// Mitsubishi GX Works2 project: project 1 auto   PLC: FX3G

// global labels: Global1
VAR_GLOBAL
  Starter AT X010 : BOOL;
  WorkDay_Lamp AT Y010 : BOOL;
  Emergancy AT X007 : BOOL;
  Invalid_Stock AT M0 : BOOL;
  Flour_Stock AT D1600 : REAL;
END_VAR
VAR_GLOBAL CONSTANT
  Const_100 : REAL := 100;
END_VAR
VAR_GLOBAL
  Yeast_Stock AT D1610 : REAL;
END_VAR
VAR_GLOBAL CONSTANT
  const_yeast_5 : REAL := 5.0;
END_VAR
VAR_GLOBAL
  Yeast_Div AT D1615 : REAL;
  Water_Stock AT D1620 : REAL;
  Water_Div AT D1625 : REAL;
END_VAR
VAR_GLOBAL CONSTANT
  Const_Water_2 : REAL := 2;
END_VAR
VAR_GLOBAL
  Oil_Stock AT D1630 : REAL;
  Oil_Div AT D1635 : REAL;
END_VAR
VAR_GLOBAL CONSTANT
  Oil_const : REAL := 3.33333333;
END_VAR
VAR_GLOBAL
  Spicies_Stock AT D1640 : REAL;
  Spicies_Div AT D1645 : REAL;
END_VAR
VAR_GLOBAL CONSTANT
  Const_Spicies_10 : REAL := 10;
  Const_3_Sec : INT := 30;
END_VAR
VAR_GLOBAL
  Start_Move AT X002 : BOOL;
  checkKK AT TS0 : BOOL;
  Lamp_Y5 AT Y005 : BOOL;
  Timer_In AT TC0 : BOOL;
END_VAR
VAR_GLOBAL CONSTANT
  TIMERINN : INT := 30;
END_VAR
VAR_GLOBAL
  check_y05 AT TS0 : BOOL;
  check_lamp5 AT M2 : BOOL;
  checkM2 AT M2 : BOOL;
  Input_X1 AT X001 : BOOL;
  Lamp_Y1 AT Y001 : BOOL;
  Start_Stage_2 AT X011 : BOOL;
  Couner_X11 AT CC2 : BOOL;
END_VAR
VAR_GLOBAL CONSTANT
  Max_11 : INT := 2;
END_VAR
VAR_GLOBAL
  Check_Counter_x11 AT CS2 : BOOL;
  Timer_Y002 AT TC1 : BOOL;
END_VAR
VAR_GLOBAL CONSTANT
  Max_Time_Y002 : INT := 10;
END_VAR
VAR_GLOBAL
  Check_Lights AT M3 : BOOL;
  Check_Y002 AT TS1 : BOOL;
  Lamp_Y2 AT Y002 : BOOL;
  Timer_Y003 AT TC2 : BOOL;
END_VAR
VAR_GLOBAL CONSTANT
  Max_Time_Y003 : INT := 10;
END_VAR
VAR_GLOBAL
  Check_Y003 AT TS2 : BOOL;
  Lamp_Y003 AT Y003 : BOOL;
END_VAR
VAR_GLOBAL CONSTANT
  Total_Time_stage2 : INT := 30;
END_VAR
VAR_GLOBAL
  Timer_Total AT TC3 : BOOL;
  Timer_Total_Ending AT TS3 : BOOL;
  Timer_Y004 AT TC4 : BOOL;
END_VAR
VAR_GLOBAL CONSTANT
  Max_Time_Y004 : INT := 40;
END_VAR
VAR_GLOBAL
  Y004_Open AT TS4 : BOOL;
  Baking_Lamp AT Y004 : BOOL;
  Check_Stage2_End AT M4 : BOOL;
  Close_Y004 AT TS4 : BOOL;
  Start_Check_Quality AT X003 : BOOL;
  Input_Analog_Value AT D8281 : REAL;
END_VAR
VAR_GLOBAL CONSTANT
  Const_2000 : DINT := 2000;
  Const_400 : DINT := 400;
END_VAR
VAR_GLOBAL
  Check_Quality_Status AT M5 : BOOL;
  Check_Quality_Value AT M5 : BOOL;
  Check_Quality_Fail AT M5 : BOOL;
  Quality_Lamp AT Y006 : BOOL;
  Check_Successful AT TS5 : BOOL;
  Check6 AT M6 : BOOL;
  Timer_Y006 AT TC5 : BOOL;
END_VAR
VAR_GLOBAL CONSTANT
  Max_Time_YOO5 : INT := 50;
END_VAR
VAR_GLOBAL
  stop_Y006 AT TS5 : BOOL;
  analog AT D8281 : WORD;
  analogResolt AT D1700 : DINT;
  y6_lamp AT Y006 : BOOL;
END_VAR
VAR_GLOBAL CONSTANT
  Max_Time_YOO6 : INT := 50;
END_VAR
VAR_GLOBAL
  Flower_Tank AT D1650 : REAL;
  Yeast_Tank AT D1655 : REAL;
  Water_Tank AT D1660 : REAL;
  Oil_Tank AT D1665 : REAL;
  Spicies_Tank AT D1670 : REAL;
  Lisha AT M1 : BOOL;
  Flower_In_Mixer AT D1675 : REAL;
  Yeast_In_Mixer AT D1680 : REAL;
  Water_In_Mixer AT D1685 : REAL;
  Oil_In_Mixer AT D1690 : REAL;
  Spicies_In_Mixer AT D1695 : REAL;
  Flower_In_Blow AT D1705 : REAL;
  Yeast_In_Blow AT D1710 : REAL;
  Water_In_Blow AT D1715 : REAL;
  Oil_In_Blow AT D1720 : REAL;
  Spicies_In_Blow AT D1725 : REAL;
END_VAR
VAR_GLOBAL CONSTANT
  Const_20 : REAL := 20;
  Const_50 : REAL := 50;
  Const_30 : REAL := 30;
  Const_10 : REAL := 10;
END_VAR
VAR_GLOBAL
  Flour_Resolt AT D1730 : REAL;
  Yeast_Result AT D1735 : REAL;
  Water_Result AT D1740 : REAL;
  Oil_Result AT D1745 : REAL;
  Spieces_Result AT D1750 : REAL;
  Flower_In_Pattern AT D1755 : REAL;
  Yeast_In_Pattern AT D1760 : REAL;
  Water_In_Pattern AT D1765 : REAL;
  Oil_In_Pattern AT D1770 : REAL;
  Spicies_In_Pattern AT D1780 : REAL;
  Counter_M5 AT CC5 : BOOL;
END_VAR
VAR_GLOBAL CONSTANT
  Max_M5 : INT := 2;
END_VAR
VAR_GLOBAL
  Drop_Pattern AT CS5 : BOOL;
  Dropping_Time AT TC6 : BOOL;
END_VAR
VAR_GLOBAL CONSTANT
  Max_Drop_Time : INT := 30;
END_VAR
VAR_GLOBAL
  Stop_Y10 AT TS6 : BOOL;
  Check_3_Lights AT M7 : BOOL;
  Timer_Y010 AT TC10 : BOOL;
END_VAR
VAR_GLOBAL CONSTANT
  Max_Time_Y010 : INT := 5;
END_VAR
VAR_GLOBAL
  stop_timerY10 AT TS10 : BOOL;
  Check_X10 AT M10 : BOOL;
  Start_Check_Quuality AT X003 : BOOL;
  Check_Light10 AT M10 : BOOL;
  Timer_Y010_Close AT TC11 : BOOL;
  Stop_3_sconds_y10 AT TS6 : BOOL;
  open_y10 AT M11 : BOOL;
  stop_timerY100 AT TS11 : BOOL;
  TRY AT M12 : BOOL;
  yosi AT M13 : BOOL;
  jwegfw AT M13 : BOOL;
  G AT M20 : BOOL;
END_VAR
VAR_GLOBAL CONSTANT
  Max_Time_Y01000 : INT := 5;
END_VAR
VAR_GLOBAL
  fictivy AT Y020 : BOOL;
  Shut_Down_Y10 AT M13 : BOOL;
  Start_New_Itaration AT M14 : BOOL;
  Invalid_Stock_Next_Itaration AT M15 : BOOL;
  notgood AT M16 : BOOL;
END_VAR

// task Task_01 (event TRUE, interval 0, priority 31): POU_01

PROGRAM POU_01
(* structured ladder/FBD written out as ST: instructions are called as NAME(EN, inputs, outputs); _pN, _eN, _tN stand for wires *)
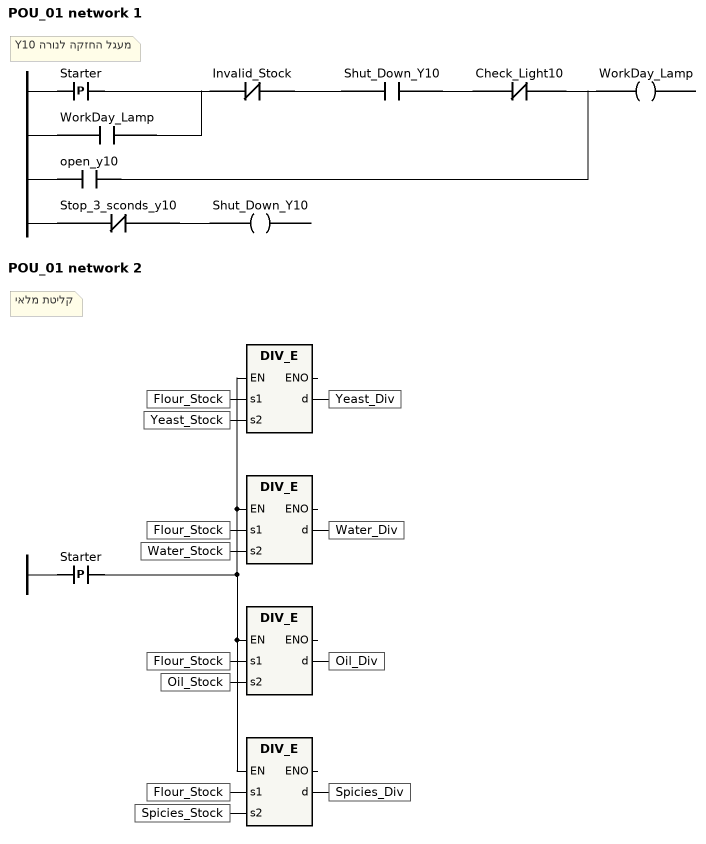
(* network 1 מעגל החזקה לנורה Y10 *)
(* מעגל החזקה לנורה Y10 *)
WorkDay_Lamp := ((((LDP(TRUE, Starter) OR WorkDay_Lamp) AND NOT Invalid_Stock) AND Shut_Down_Y10) AND NOT Check_Light10) OR open_y10;
Shut_Down_Y10 := NOT Stop_3_sconds_y10;
(* network 2 קליטת וחישוב מלאי *)
(* קליטת מלאי *)
_p1 := LDP(TRUE, Starter);
DIV_E(_p1, Flour_Stock, Yeast_Stock, Yeast_Div);
DIV_E(_p1, Flour_Stock, Water_Stock, Water_Div);
DIV_E(_p1, Flour_Stock, Oil_Stock, Oil_Div);
DIV_E(_p1, Flour_Stock, Spicies_Stock, Spicies_Div);
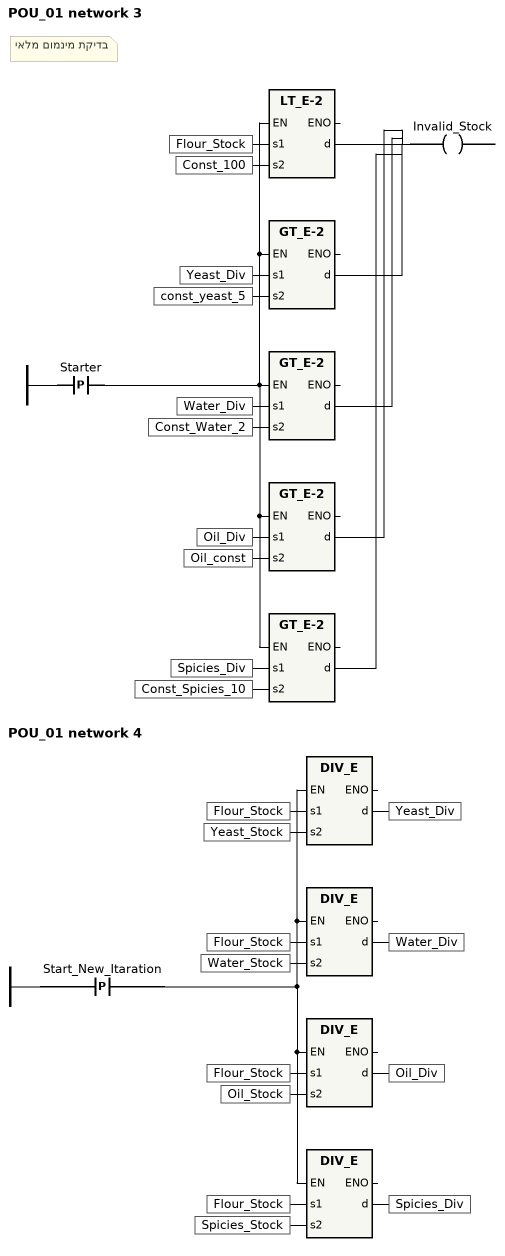
(* network 3 בדיקת מינימום מלאי *)
(* בדיקת מינמום מלאי *)
_p1 := LDP(TRUE, Starter);
LT_E(_p1, Flour_Stock, Const_100, _t2);
GT_E(_p1, Yeast_Div, const_yeast_5, _t3);
GT_E(_p1, Water_Div, Const_Water_2, _t4);
GT_E(_p1, Oil_Div, Oil_const, _t5);
GT_E(_p1, Spicies_Div, Const_Spicies_10, _t6);
Invalid_Stock := _t2 OR _t3 OR _t4 OR _t5 OR _t6;
(* network 4 בדיקת מלאי נוספת *)
_p1 := LDP(TRUE, Start_New_Itaration);
DIV_E(_p1, Flour_Stock, Yeast_Stock, Yeast_Div);
DIV_E(_p1, Flour_Stock, Water_Stock, Water_Div);
DIV_E(_p1, Flour_Stock, Oil_Stock, Oil_Div);
DIV_E(_p1, Flour_Stock, Spicies_Stock, Spicies_Div);
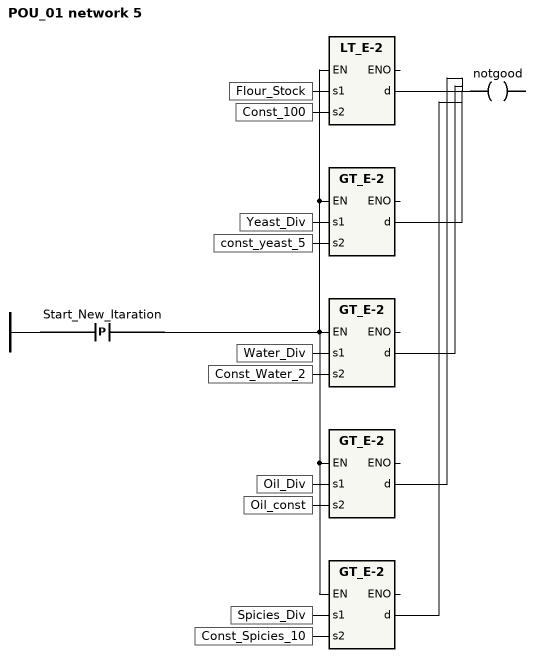
(* network 5 בדיקת מלאי נוספת *)
_p1 := LDP(TRUE, Start_New_Itaration);
LT_E(_p1, Flour_Stock, Const_100, _t2);
GT_E(_p1, Yeast_Div, const_yeast_5, _t3);
GT_E(_p1, Water_Div, Const_Water_2, _t4);
GT_E(_p1, Oil_Div, Oil_const, _t5);
GT_E(_p1, Spicies_Div, Const_Spicies_10, _t6);
notgood := _t2 OR _t3 OR _t4 OR _t5 OR _t6;
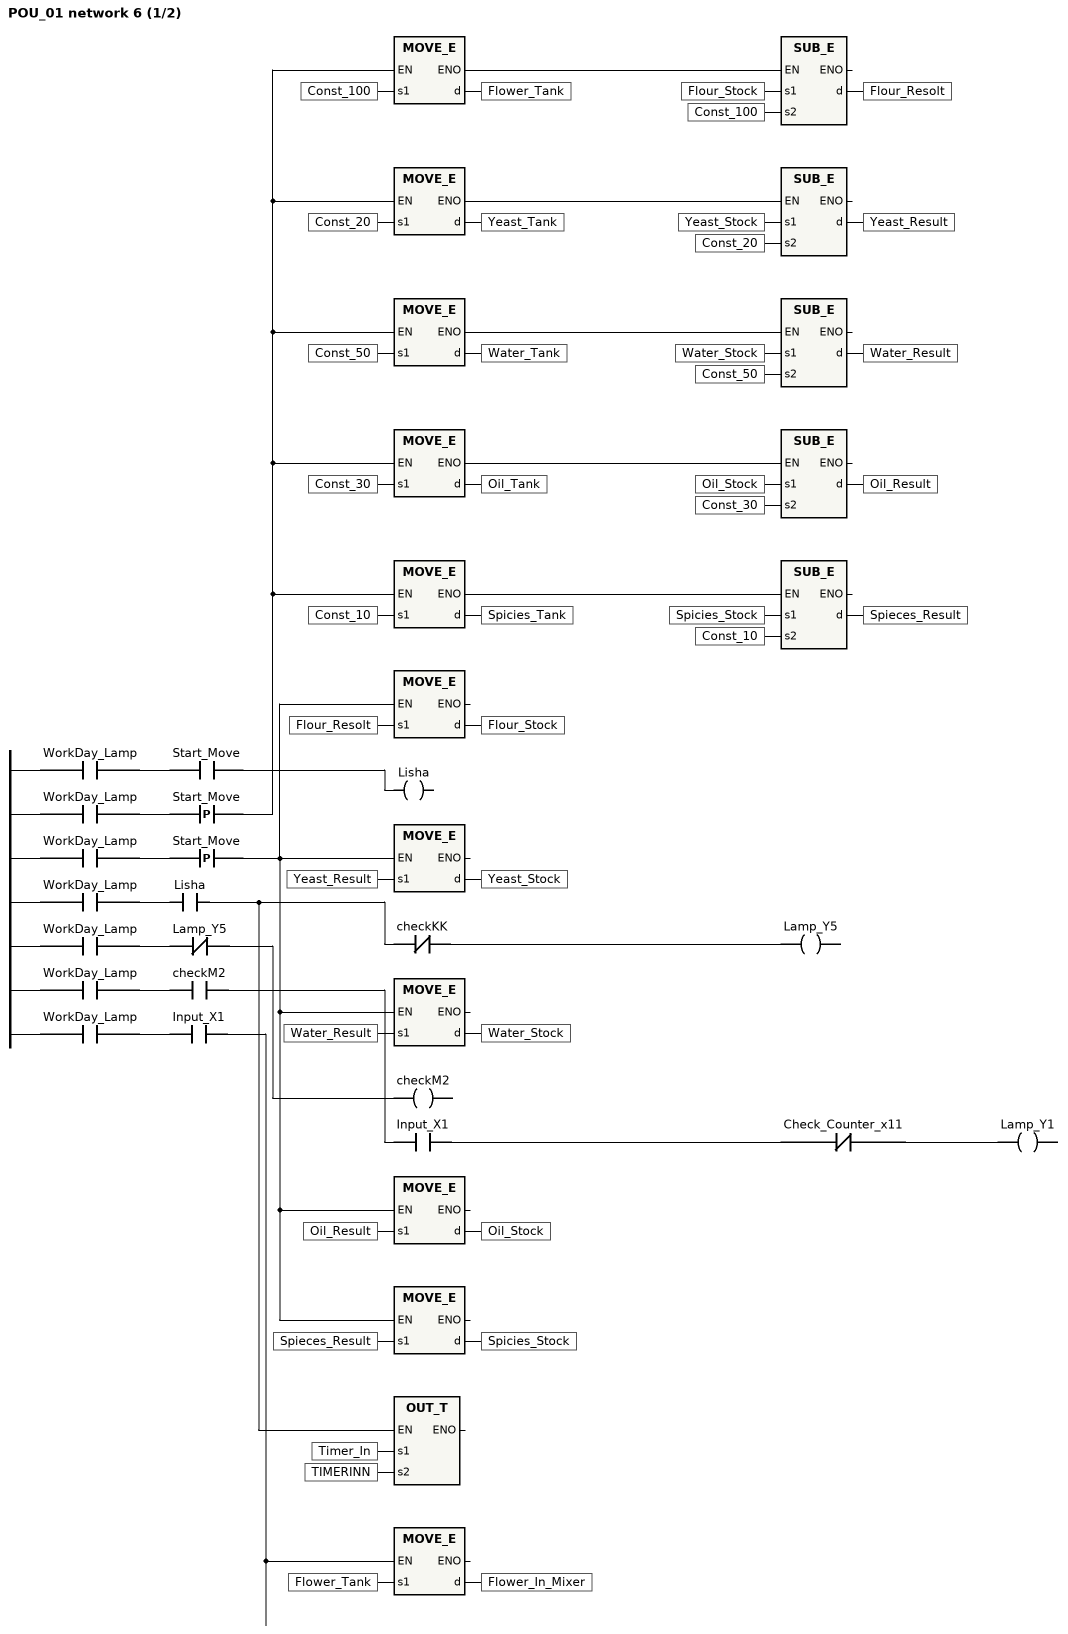
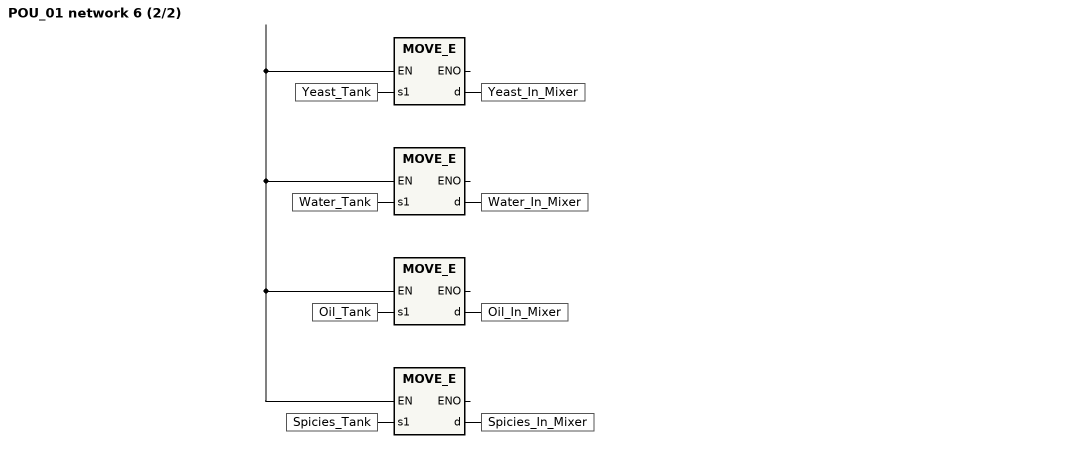
(* network 6 שלב 1  *)
Lisha := WorkDay_Lamp AND Start_Move;
_p1 := WorkDay_Lamp AND LDP(TRUE, Start_Move);
_e2 := MOVE_E(_p1, Const_100, Flower_Tank);
SUB_E(_e2, Flour_Stock, Const_100, Flour_Resolt);
_e3 := MOVE_E(_p1, Const_20, Yeast_Tank);
SUB_E(_e3, Yeast_Stock, Const_20, Yeast_Result);
_e4 := MOVE_E(_p1, Const_50, Water_Tank);
SUB_E(_e4, Water_Stock, Const_50, Water_Result);
_e5 := MOVE_E(_p1, Const_30, Oil_Tank);
SUB_E(_e5, Oil_Stock, Const_30, Oil_Result);
_e6 := MOVE_E(_p1, Const_10, Spicies_Tank);
SUB_E(_e6, Spicies_Stock, Const_10, Spieces_Result);
_p7 := WorkDay_Lamp AND LDP(TRUE, Start_Move);
MOVE_E(_p7, Flour_Resolt, Flour_Stock);
MOVE_E(_p7, Yeast_Result, Yeast_Stock);
MOVE_E(_p7, Water_Result, Water_Stock);
MOVE_E(_p7, Oil_Result, Oil_Stock);
MOVE_E(_p7, Spieces_Result, Spicies_Stock);
_p8 := WorkDay_Lamp AND Lisha;
OUT_T(_p8, Timer_In, TIMERINN);
Lamp_Y5 := _p8 AND NOT checkKK;
checkM2 := WorkDay_Lamp AND NOT Lamp_Y5;
Lamp_Y1 := WorkDay_Lamp AND checkM2 AND Input_X1 AND NOT Check_Counter_x11;
_p9 := WorkDay_Lamp AND Input_X1;
MOVE_E(_p9, Flower_Tank, Flower_In_Mixer);
MOVE_E(_p9, Yeast_Tank, Yeast_In_Mixer);
MOVE_E(_p9, Water_Tank, Water_In_Mixer);
MOVE_E(_p9, Oil_Tank, Oil_In_Mixer);
MOVE_E(_p9, Spicies_Tank, Spicies_In_Mixer);
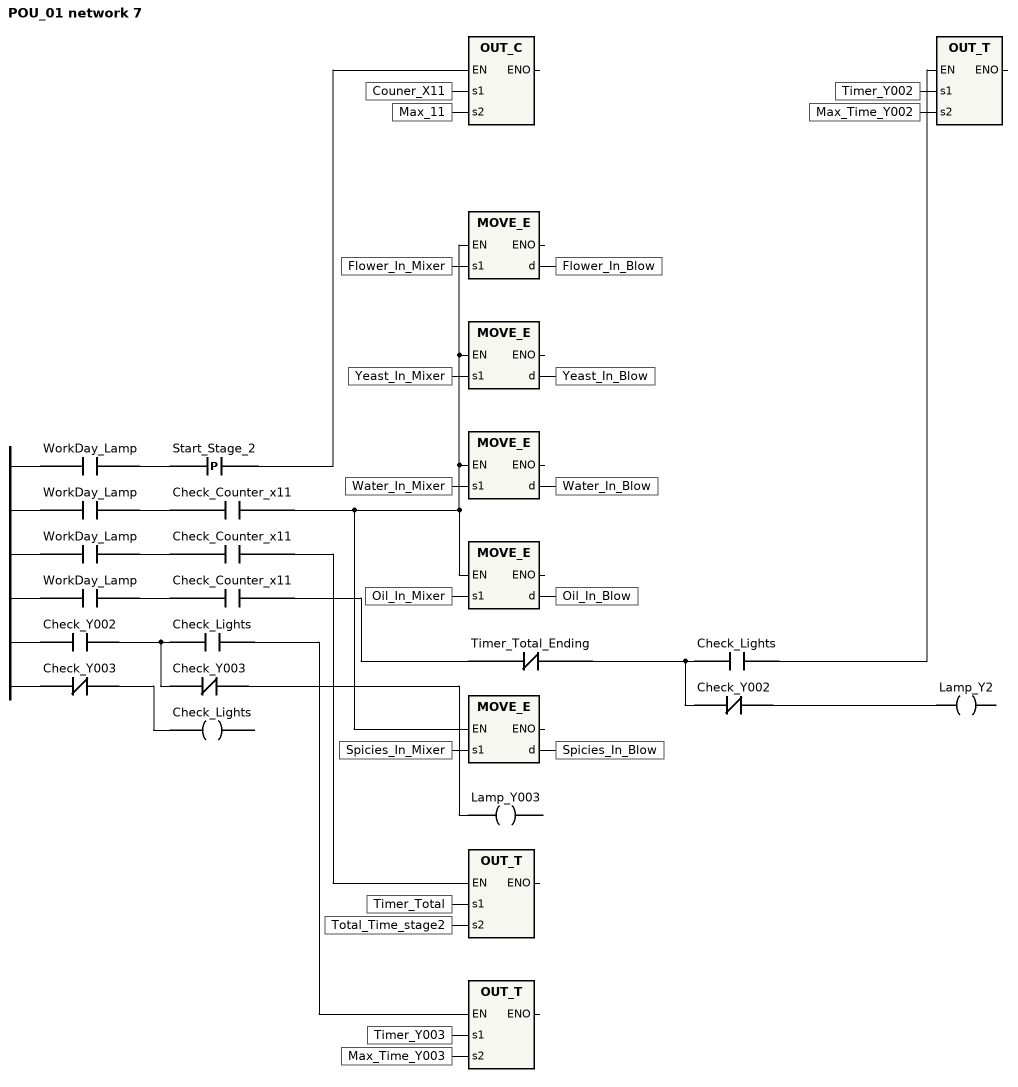
(* network 7 שלב 2 *)
OUT_C(WorkDay_Lamp AND LDP(TRUE, Start_Stage_2), Couner_X11, Max_11);
_p1 := WorkDay_Lamp AND Check_Counter_x11;
MOVE_E(_p1, Flower_In_Mixer, Flower_In_Blow);
MOVE_E(_p1, Yeast_In_Mixer, Yeast_In_Blow);
MOVE_E(_p1, Water_In_Mixer, Water_In_Blow);
MOVE_E(_p1, Oil_In_Mixer, Oil_In_Blow);
MOVE_E(_p1, Spicies_In_Mixer, Spicies_In_Blow);
OUT_T(WorkDay_Lamp AND Check_Counter_x11, Timer_Total, Total_Time_stage2);
_p2 := WorkDay_Lamp AND Check_Counter_x11 AND NOT Timer_Total_Ending;
OUT_T(_p2 AND Check_Lights, Timer_Y002, Max_Time_Y002);
Lamp_Y2 := _p2 AND NOT Check_Y002;
OUT_T(Check_Y002 AND Check_Lights, Timer_Y003, Max_Time_Y003);
Lamp_Y003 := Check_Y002 AND NOT Check_Y003;
Check_Lights := NOT Check_Y003;
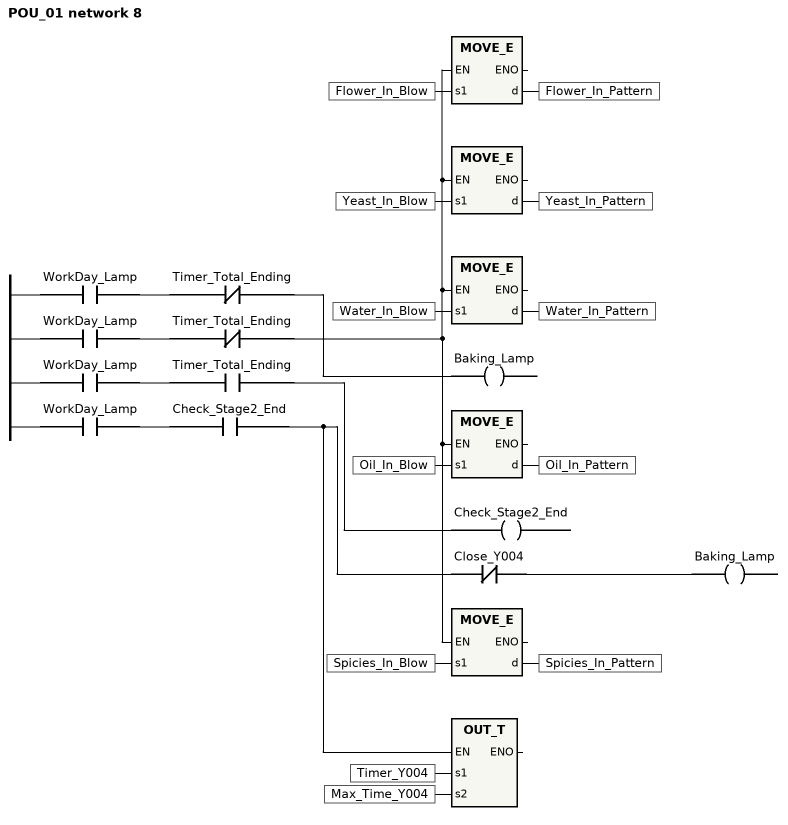
(* network 8 שלב 3 *)
Baking_Lamp := WorkDay_Lamp AND NOT Timer_Total_Ending;
_p1 := WorkDay_Lamp AND NOT Timer_Total_Ending;
MOVE_E(_p1, Flower_In_Blow, Flower_In_Pattern);
MOVE_E(_p1, Yeast_In_Blow, Yeast_In_Pattern);
MOVE_E(_p1, Water_In_Blow, Water_In_Pattern);
MOVE_E(_p1, Oil_In_Blow, Oil_In_Pattern);
MOVE_E(_p1, Spicies_In_Blow, Spicies_In_Pattern);
Check_Stage2_End := WorkDay_Lamp AND Timer_Total_Ending;
_p2 := WorkDay_Lamp AND Check_Stage2_End;
OUT_T(_p2, Timer_Y004, Max_Time_Y004);
Baking_Lamp := _p2 AND NOT Close_Y004;
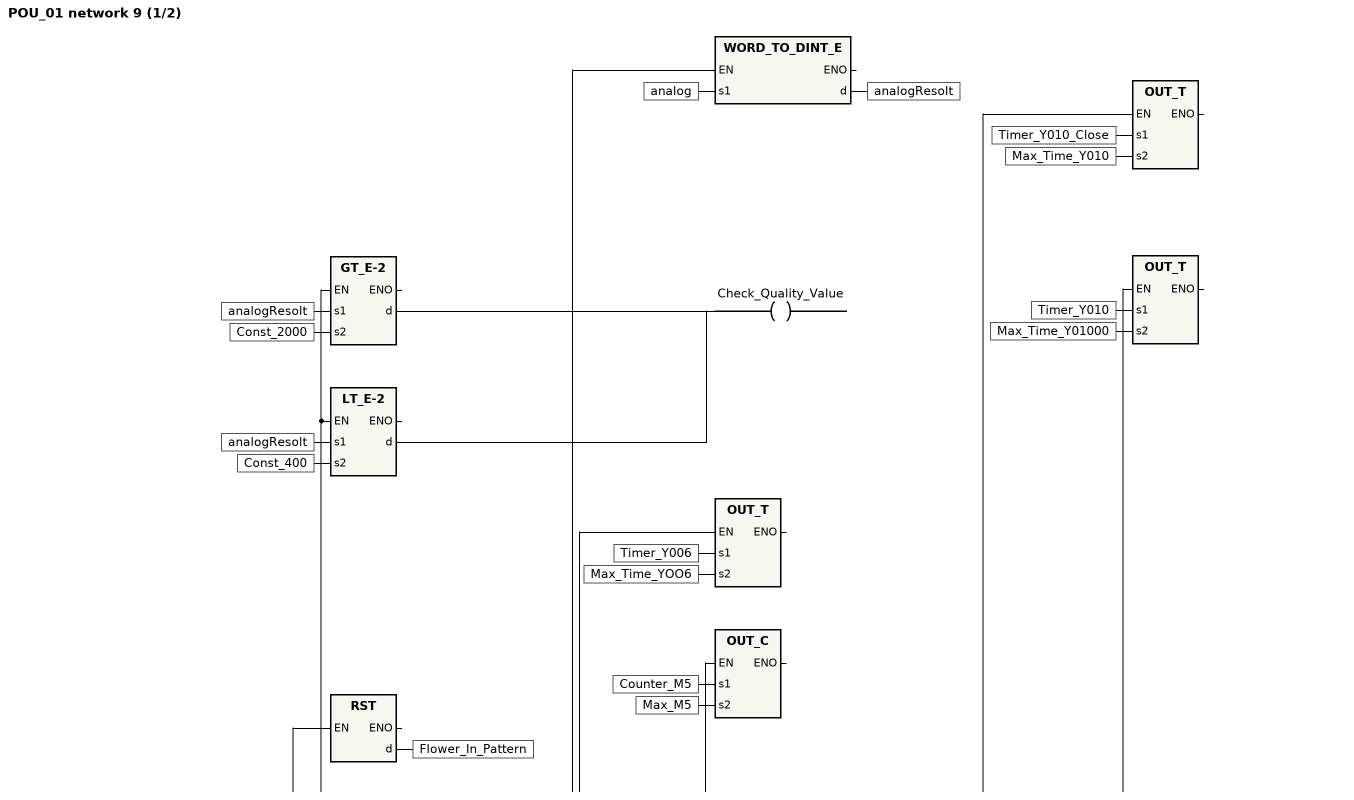
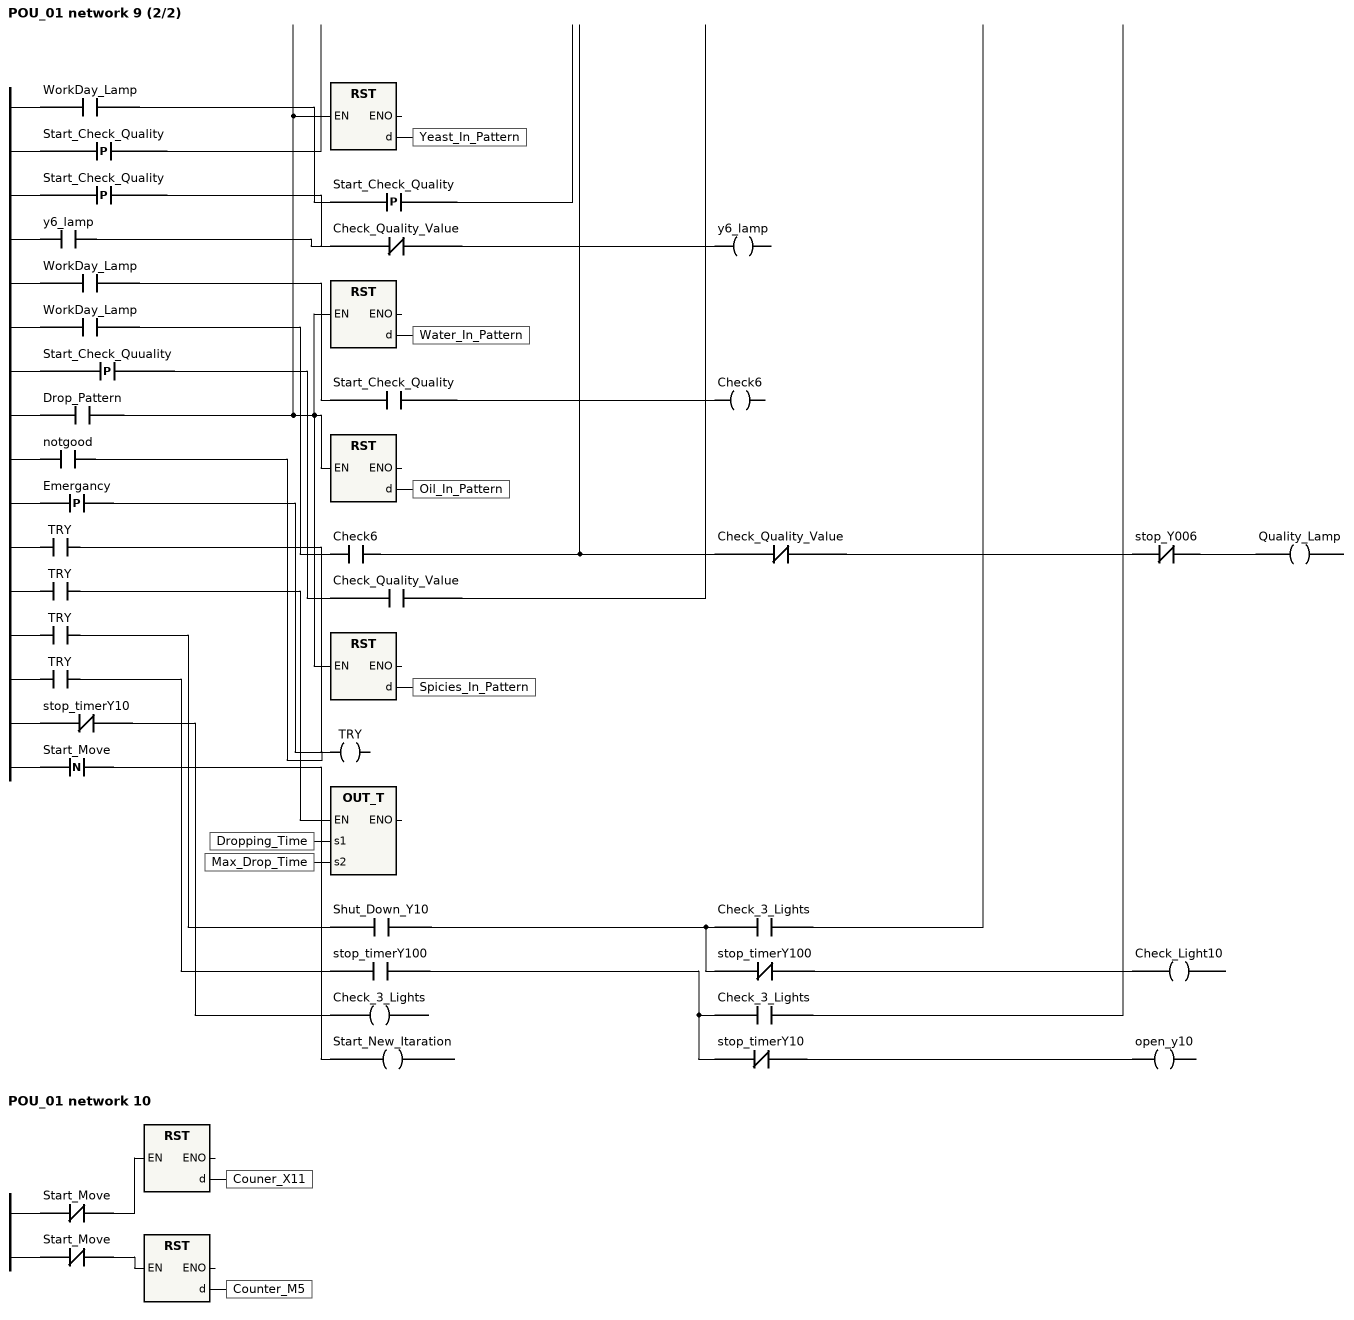
(* network 9 שלב 4 *)
WORD_TO_DINT_E(WorkDay_Lamp AND LDP(TRUE, Start_Check_Quality), analog, analogResolt);
_p1 := LDP(TRUE, Start_Check_Quality);
GT_E(_p1, analogResolt, Const_2000, _t2);
LT_E(_p1, analogResolt, Const_400, _t3);
Check_Quality_Value := _t2 OR _t3;
y6_lamp := (LDP(TRUE, Start_Check_Quality) OR y6_lamp) AND NOT Check_Quality_Value;
Check6 := WorkDay_Lamp AND Start_Check_Quality;
_p4 := WorkDay_Lamp AND Check6;
OUT_T(_p4, Timer_Y006, Max_Time_YOO6);
Quality_Lamp := _p4 AND NOT Check_Quality_Value AND NOT stop_Y006;
OUT_C(LDP(TRUE, Start_Check_Quuality) AND Check_Quality_Value, Counter_M5, Max_M5);
RST(Drop_Pattern, Flower_In_Pattern);
RST(Drop_Pattern, Yeast_In_Pattern);
RST(Drop_Pattern, Water_In_Pattern);
RST(Drop_Pattern, Oil_In_Pattern);
RST(Drop_Pattern, Spicies_In_Pattern);
TRY := notgood OR LDP(TRUE, Emergancy) OR TRY;
OUT_T(TRY, Dropping_Time, Max_Drop_Time);
_p5 := TRY AND Shut_Down_Y10;
OUT_T(_p5 AND Check_3_Lights, Timer_Y010_Close, Max_Time_Y010);
Check_Light10 := _p5 AND NOT stop_timerY100;
_p6 := TRY AND stop_timerY100;
OUT_T(_p6 AND Check_3_Lights, Timer_Y010, Max_Time_Y01000);
open_y10 := _p6 AND NOT stop_timerY10;
Check_3_Lights := NOT stop_timerY10;
Start_New_Itaration := LDF(TRUE, Start_Move);
(* network 10 *)
RST(NOT Start_Move, Couner_X11);
RST(NOT Start_Move, Counter_M5);
END_PROGRAM
